FUNCTION_BLOCK F_ACCUM_LREAL (* Used for accumulating data. Reset to INIT using R event. *)
  (* Standard: 61499-2 *)
  (* Version 1.1, 2017-06-14, Marc Jakobi, HTW Berlin *)
  (* Version 1.0, 2016-05-26, AZ, fortiss GmbH *)
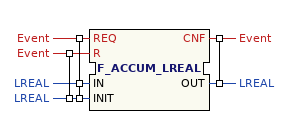
  EVENT_INPUT
    REQ WITH IN, INIT; (* Normal Execution Request *)
    R WITH INIT; (* Reset *)
  END_EVENT
  EVENT_OUTPUT
    CNF WITH OUT; (* Execution Confirmation *)
  END_EVENT
  VAR_INPUT
    IN : LREAL; (* Value to accumulate *)
    INIT : LREAL; (* Initial value *)
  END_VAR
  VAR_OUTPUT
    OUT : LREAL; (* Accumulated value *)
  END_VAR
  VAR
    CACHE : LREAL; (* Internal Variable *)
  END_VAR
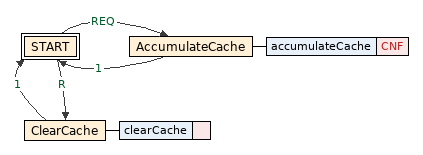
  EC_STATES
    START;
    AccumulateCache : accumulateCache -> CNF; (* Normal execution *)
    ClearCache : clearCache;
  END_STATES
  EC_TRANSITIONS
    START TO AccumulateCache := REQ;
    AccumulateCache TO START := 1;
    START TO ClearCache := R;
    ClearCache TO START := 1;
  END_TRANSITIONS
  ALGORITHM accumulateCache IN ST: (* Accumulates time *)
CACHE  := CACHE + IN;
OUT := CACHE;
  END_ALGORITHM
  ALGORITHM clearCache IN ST: (* Resets internal memory to INIT input *)
CACHE := INIT;
  END_ALGORITHM
END_FUNCTION_BLOCK
